(* PLC project static_torsion.project, CODESYS CODESYS V3.5 SP17 Patch 3 *)
(* stored: creationDateTime 1970-01-01T00:00:00, modificationDateTime 2026-06-22T15:12:39.4699931 *)

(* {attribute 'strict'} *)
{attribute 'qualified_only'}
TYPE CTRL_ID : (POWER_OFF := 0, POWER_ON := 1, ERROR_RESET := 2, MOVE_REL := 3, JOG_FWD := 4, JOG_BACK := 5, MOVE_FOLLOW := 6, HALT := 7, STOP := 100) UINT;
END_TYPE
